# EPICS StreamDevice protocol: examples/07_stream/demoApp/Db/si.proto
# Stream Protocol file for simpleInstrument.py

Terminator = CR LF;
InTerminator = CR LF;
ReplyTimeout = 10000;
ReadTimeout = 10000;

getVolt
{
  out "VOLTS?";
  in "VOLTS %f";
}

setVolt
{
  out "VOLTS %f";
  @init
  {
    getVolt;
  }
}

getCurr
{
  out "CURR?";
  in "CURR %f";
}
